TYPE ST_StepSequencer :
STRUCT
	bStep					: ARRAY [0..63] OF BOOL;  		//Game Play Sequence Step number trigger
END_STRUCT
END_TYPE

(* stored: Version 1.1.0.1, ProductVersion 3.1.4024.10
   DUT ST_StepSequencer: Id {abed617c-cf01-4ee9-928d-6b8189da4dd6} *)
